TYPE ST_MyType :
STRUCT
	bValue	: BOOL;
	iValue	: INT;
	sValue	: STRING;
END_STRUCT
END_TYPE

(* stored: Version 1.1.0.1, ProductVersion 3.1.4024.12
   DUT ST_MyType: Id {e063907c-5260-473f-ad6a-6a0cd6695c22} *)
